(* IEC 61131-3 sources: ArfBotOS/Codesys-4/ArfBotOS.fbsdev/Application.iecapp^/FUN/vision/FB_VisionCmdProcessor.fb.st^/public, 1 file *)

(* ---- M_ReconnectVisionSystem.meth.st ---- *)
METHOD PUBLIC M_ReconnectVisionSystem : BOOL
VAR_INPUT
END_VAR

// TODO may want to make sure the state machine is not in execute?
_Vision.M_Reconnect();
END_METHOD
